DATA_BLOCK "DB"
{ S7_Optimized_Access := 'true' }
    VAR
        timer_t: LREAL;
        timer: DINT;
        sup: DINT;
        hw_button_bit: BOOL;
        hw_button: DINT;
        hw_lamp_bit: BOOL;
        hw_lamp: DINT;
        firstRun: BOOL;
        curTimer: INT;
    END_VAR
BEGIN
    firstRun := TRUE;
END_DATA_BLOCK
